Yaskawa INFORM job: X2_242(90,180).JBI

/JOB
//NAME X2_242(90,180)
///FOLDERNAME X2
//POS
///NPOS 135,135,135,3,0,0
///TOOL 0
///POSTYPE PULSE
///PULSE
C00000=-2000,-130321,-133031,0,28968,0
C00001=-117091,-130321,-133031,2123,28968,-3391
C00002=-159919,-130321,-133031,2123,28968,-3391
C00003=-159919,-130321,-133031,2123,87939,-3391
C00004=-105022,-108859,-78959,-31083,72176,-68730
C00005=-151007,-25092,-39063,-12800,65605,78235
C00006=-132593,67036,12002,-14068,96381,18620
C00007=-133669,66493,21901,-13656,90017,18991
C00008=-134090,67791,24612,-13544,88977,18967
C00009=-134090,67273,25686,-13543,88075,19066
C00010=-134090,67791,24612,-13544,88977,18967
C00011=-134073,67330,25416,-13547,88268,19050
C00012=-134739,69521,27996,-13380,87713,18892
C00013=-134073,67330,25416,-13547,88268,19050
C00014=-132576,62954,16151,-13952,91863,19138
C00015=-158058,56370,5063,-6789,93126,-12165
C00016=-161492,61731,13256,-13118,78465,-26852
C00017=-161219,65846,21027,-13360,75906,-26484
C00018=-161113,67624,24299,-13466,74851,-26332
C00019=-161114,67102,25367,-13521,73950,-26231
C00020=-161163,66904,24770,-13484,74201,-26276
C00021=-160433,68822,27026,-13824,73925,-25997
C00022=-161163,66904,24770,-13484,74201,-26276
C00023=-161111,67182,25269,-13516,74049,-26241
C00024=-161656,69750,28292,-13313,73437,-26358
C00025=-161111,67182,25269,-13516,74049,-26241
C00026=-161490,61134,14077,-13154,77673,-26766
C00027=-156757,36958,-7461,-10431,80488,-32893
C00028=-156267,40068,-956,-10702,78181,-32538
C00029=-156253,41350,1581,-10739,77295,-32458
C00030=-163911,62406,19268,6086,89764,-33901
C00031=-164446,59700,16177,9989,92313,-36673
C00032=-164418,59610,16075,9984,92326,-36663
C00033=-161961,50915,7130,7396,91423,-24195
C00034=-156779,43944,226,1104,89071,-15308
C00035=-150790,45819,2072,-7115,89912,-6230
C00036=-145239,57854,15312,-8608,88471,-4374
C00037=-145092,58025,15712,-8678,88333,-4325
C00038=-139841,72267,32142,-17294,91315,7524
C00039=-140946,99356,62874,-12757,94092,30974
C00040=-141208,101673,65869,-12719,93415,30955
C00041=-122713,94046,59869,-28177,93377,67521
C00042=-121487,97083,60557,-28349,94790,67637
C00043=-133468,48615,1742,-18804,93124,11842
C00044=-157997,71741,26694,-3661,70569,-66185
C00045=-156653,80960,41725,-4466,66130,-65572
C00046=-160707,58811,27097,7838,50776,-65613
C00047=-161862,58527,28132,10661,48808,-66136
C00048=-162060,71887,38599,9565,55625,-66013
C00049=-162634,67727,36532,11016,51381,-65293
C00050=-160821,61019,33044,3636,43624,-62105
C00051=-154148,75334,40185,-14517,57905,-63097
C00052=-154196,71820,32295,-14055,60854,-63507
C00053=-153288,55034,31796,-23088,50010,-69293
C00054=-151031,57353,45940,-40148,40347,-64995
C00055=-150621,58129,46816,-40537,40429,-64769
C00056=-149751,55668,48450,-47014,34319,-61006
C00057=-150747,54467,47461,-43008,31230,-60446
C00058=-154056,49858,42858,-29251,25609,-68749
C00059=-154872,47959,37614,-21306,28921,-70888
C00060=-159207,48403,28271,-1768,40383,-74494
C00061=-149846,52946,33243,-13952,46682,-81563
C00062=-149940,61587,46564,-14806,43022,-81015
C00063=-146336,59430,51340,-33146,36492,-77110
C00064=-145282,69746,63346,-35645,35179,-75711
C00065=-143319,74757,70706,-41882,34093,-73425
C00066=-141946,81470,79320,-45365,33350,-71705
C00067=-140704,87470,87386,-49528,32633,-69847
C00068=-140891,72507,62697,-35215,38758,-74780
C00069=-145179,75875,59784,-18821,43244,-78638
C00070=-151007,-25092,-39063,-12800,65605,78235
C00071=-105022,-108859,-78959,-31083,72176,-68730
C00072=-159919,-130321,-133031,2123,87939,-3391
C00073=-159919,-130321,-133031,2123,28968,-3391
C00074=-117091,-130321,-133031,2123,28968,-3391
C00075=31465,-130321,-133031,2123,28968,-3391
C00076=31465,-130321,-133031,2123,28968,-3391
C00077=70388,-93367,-87979,22259,92531,-40632
C00078=132234,14944,-6259,12342,59781,-23208
C00079=146205,63473,16177,10072,90044,-15024
C00080=148576,68007,22640,9405,88157,-14412
C00081=148576,67267,23954,9407,86985,-14500
C00082=148576,66783,24956,9411,86132,-14562
C00083=148576,66832,24863,9408,86216,-14555
C00084=149047,69084,27509,9276,85699,-14442
C00085=148423,68574,25700,9447,86607,-14574
C00086=146195,62986,16971,10071,89317,-15086
C00087=176137,58081,9771,-3198,80109,33161
C00088=174052,65626,21441,-2357,76742,32574
C00089=173571,63404,20046,-2157,76447,32425
C00090=173571,63211,20421,-2158,76117,32429
C00091=173571,63292,20263,-2157,76255,32427
C00092=172556,64401,21545,-1729,76012,32099
C00093=173019,62971,18478,-1917,77173,32231
C00094=167045,54371,14180,12829,67421,32117
C00095=167300,57261,17419,12739,66888,32149
C00096=166775,56105,16119,12998,67167,31995
C00097=174959,61653,15361,-2721,78467,32830
C00098=153862,58220,7137,12336,84382,31788
C00099=154888,58914,9595,11964,83110,31986
C00100=146416,53637,12500,29969,73855,35683
C00101=161804,89703,42514,-6671,93266,37768
C00102=160481,83040,34267,-6425,94812,37264
C00103=160461,82996,34213,-6421,94821,37257
C00104=160314,82402,33477,-6393,94958,37204
C00105=155818,71683,20777,1425,95566,24197
C00106=154068,75736,24755,2435,97986,16967
C00107=150406,78568,28210,7412,98870,8330
C00108=143192,78361,31098,15429,92978,3071
C00109=142524,84239,37703,11837,92418,-12035
C00110=142502,84415,37922,11841,92377,-12046
C00111=137937,102743,61702,17663,90401,-30375
C00112=138214,107970,68255,17604,89055,-30475
C00113=138254,108650,69203,17597,88823,-30493
C00114=137728,105908,62856,17713,91318,-30315
C00115=129809,68648,23314,23742,79294,-62187
C00116=130521,38108,-11366,22924,75116,-53839
C00117=144715,56131,10361,11744,72134,27543
C00118=151566,59831,28742,-2859,46138,64220
C00119=152051,66365,37606,-3402,44065,64516
C00120=152470,67516,39026,-3796,43800,64724
C00121=153239,74187,48057,-1867,40213,65616
C00122=151811,68486,39030,4846,43626,66812
C00123=148976,61300,30711,7226,45253,65595
C00124=147729,58500,33654,14300,37151,64277
C00125=144430,59667,36614,25817,36412,63257
C00126=144460,72482,45840,17180,42284,64323
C00127=143111,63918,40413,22730,36091,62179
C00128=143801,66633,41900,20305,38275,63153
C00129=139817,77107,57238,29606,33210,58883
C00130=141383,82478,55565,14874,41935,61497
C00131=144692,57703,21103,13544,52726,73165
C00132=140496,9250,-2578,20724,48099,77689
C00133=103999,-84119,-66645,26288,35960,55555
C00134=-2000,-130321,-133031,0,28968,0
BC00000=147972,491577,1075193
BC00001=188398,1906,1075193
BC00002=367644,-164195,1075193
BC00003=367644,-172087,1075193
BC00004=367644,-179096,239389
BC00005=367644,-179096,202799
BC00006=311795,-165148,45027
BC00007=311795,-165148,45027
BC00008=311795,-165148,45027
BC00009=311795,-165148,45027
BC00010=311795,-165148,45027
BC00011=311795,-165148,45027
BC00012=311795,-165148,45027
BC00013=311795,-165148,45027
BC00014=311795,-165148,45027
BC00015=362414,-140809,31779
BC00016=380271,-154677,8218
BC00017=380271,-154677,8218
BC00018=380271,-154677,8218
BC00019=380271,-154677,8218
BC00020=380271,-154677,8218
BC00021=380271,-154677,8218
BC00022=380271,-154677,8218
BC00023=380271,-154677,8218
BC00024=380271,-154677,8218
BC00025=380271,-154677,8218
BC00026=380271,-154677,8218
BC00027=343072,-138712,53288
BC00028=343072,-138712,53288
BC00029=343072,-138712,53288
BC00030=343072,-138712,53288
BC00031=343072,-138713,53287
BC00032=343072,-138713,53287
BC00033=343072,-138712,53288
BC00034=343072,-138712,53286
BC00035=343072,-138712,53286
BC00036=343072,-138712,53286
BC00037=343072,-138712,53284
BC00038=343072,-138712,53286
BC00039=343072,-138712,53286
BC00040=343072,-138712,53286
BC00041=294648,-138712,53288
BC00042=294648,-138712,53288
BC00043=320422,-160767,40892
BC00044=369045,-176137,27013
BC00045=367905,-178617,27013
BC00046=367905,-178910,27013
BC00047=367905,-178910,27013
BC00048=367905,-179959,27013
BC00049=367905,-180015,27013
BC00050=367905,-179162,27013
BC00051=367905,-179037,27013
BC00052=367905,-178812,27013
BC00053=384322,-166528,125648
BC00054=384322,-166528,125648
BC00055=384322,-166528,125648
BC00056=384322,-166528,125648
BC00057=384322,-166528,125648
BC00058=384322,-166528,125648
BC00059=384322,-166528,125648
BC00060=384322,-166528,125648
BC00061=367644,-168516,156611
BC00062=367644,-172191,156611
BC00063=367644,-171321,156611
BC00064=367644,-179096,156611
BC00065=367644,-179096,156611
BC00066=367644,-179096,156611
BC00067=367644,-179096,156611
BC00068=367644,-179096,156611
BC00069=367644,-179096,156611
BC00070=367644,-179096,202799
BC00071=367644,-179096,239389
BC00072=367644,-179096,1075193
BC00073=367644,-179096,1075193
BC00074=188398,1906,1075193
BC00075=341060,491577,1075193
BC00076=341060,491577,1075193
BC00077=258990,522046,241931
BC00078=356760,522046,241931
BC00079=356760,409759,42887
BC00080=356760,409759,42887
BC00081=356760,409759,42887
BC00082=356760,409759,42887
BC00083=356760,409759,42887
BC00084=356760,409759,42887
BC00085=356760,409759,42887
BC00086=356760,409759,42887
BC00087=398158,391605,17411
BC00088=398158,391605,17411
BC00089=398158,391605,17411
BC00090=398158,391605,17411
BC00091=398158,391605,17411
BC00092=398158,391605,17411
BC00093=398158,391605,17411
BC00094=398158,391605,17411
BC00095=398158,391605,17411
BC00096=398158,391605,17411
BC00097=398158,391605,17411
BC00098=344176,409815,17
BC00099=344176,409815,17
BC00100=344176,409815,17
BC00101=344176,409815,17
BC00102=344176,409815,17
BC00103=344176,409815,17
BC00104=344176,409815,17
BC00105=344176,409815,15
BC00106=344176,409815,17
BC00107=344176,409815,17
BC00108=344176,409815,13
BC00109=344176,409815,12
BC00110=344176,409815,12
BC00111=344176,409815,12
BC00112=344176,409815,12
BC00113=344176,409815,12
BC00114=344176,409815,12
BC00115=326504,409815,17
BC00116=326504,409815,17
BC00117=339270,441939,17014
BC00118=344994,456339,24633
BC00119=344994,456339,24633
BC00120=344994,456339,24633
BC00121=344994,456339,24633
BC00122=344994,456339,24631
BC00123=344994,456339,24631
BC00124=344994,456339,24631
BC00125=344994,456339,24631
BC00126=344994,456339,24631
BC00127=344994,456339,24631
BC00128=344994,456339,24631
BC00129=344994,456339,24631
BC00130=344994,456339,24631
BC00131=359830,449275,49809
BC00132=372188,522287,309305
BC00133=335727,515780,471592
BC00134=200118,491577,1075193
EC00000=-798156,-1296783
EC00001=-798156,-1296783
EC00002=-798156,-1296783
EC00003=-798156,-1296783
EC00004=-798156,-1296783
EC00005=-798156,-1296783
EC00006=-798156,-1296783
EC00007=-798156,-1296783
EC00008=-798156,-1296783
EC00009=-798156,-1296783
EC00010=-798156,-1296783
EC00011=-798156,-1296783
EC00012=-798156,-1296783
EC00013=-798156,-1296783
EC00014=-798156,-1296783
EC00015=-798156,-1296783
EC00016=-798156,-1296783
EC00017=-798156,-1296783
EC00018=-798156,-1296783
EC00019=-798156,-1296783
EC00020=-798156,-1296783
EC00021=-798156,-1296783
EC00022=-798156,-1296783
EC00023=-798156,-1296783
EC00024=-798156,-1296783
EC00025=-798156,-1296783
EC00026=-798156,-1296783
EC00027=-798156,-1296783
EC00028=-798156,-1296783
EC00029=-798156,-1296783
EC00030=-798156,-1296783
EC00031=-798155,-1296782
EC00032=-798155,-1296782
EC00033=-798156,-1296783
EC00034=-798155,-1296782
EC00035=-798155,-1296782
EC00036=-798155,-1296782
EC00037=-798155,-1296781
EC00038=-798155,-1296782
EC00039=-798155,-1296782
EC00040=-798155,-1296782
EC00041=-798156,-1296783
EC00042=-798156,-1296783
EC00043=-798156,-1296783
EC00044=-798156,-1296783
EC00045=-798156,-1296783
EC00046=-798156,-1296783
EC00047=-798156,-1296783
EC00048=-798156,-1296783
EC00049=-798156,-1296783
EC00050=-798156,-1296783
EC00051=-798156,-1296783
EC00052=-798156,-1296783
EC00053=-798156,-1296783
EC00054=-798156,-1296783
EC00055=-798156,-1296783
EC00056=-798156,-1296783
EC00057=-798156,-1296783
EC00058=-798156,-1296783
EC00059=-798156,-1296783
EC00060=-798156,-1296783
EC00061=-798156,-1296783
EC00062=-798156,-1296783
EC00063=-798156,-1296783
EC00064=-798156,-1296783
EC00065=-798156,-1296783
EC00066=-798156,-1296783
EC00067=-798156,-1296783
EC00068=-798156,-1296783
EC00069=-798156,-1296783
EC00070=-798156,-1296783
EC00071=-798156,-1296783
EC00072=-798156,-1296783
EC00073=-798156,-1296783
EC00074=-798156,-1296783
EC00075=-798156,-1296783
EC00076=798156,-1296783
EC00077=798156,-1296783
EC00078=798156,-1296783
EC00079=798156,-1296783
EC00080=798156,-1296783
EC00081=798156,-1296783
EC00082=798156,-1296783
EC00083=798156,-1296783
EC00084=798156,-1296783
EC00085=798156,-1296783
EC00086=798156,-1296783
EC00087=798156,-1296783
EC00088=798156,-1296783
EC00089=798156,-1296783
EC00090=798156,-1296783
EC00091=798156,-1296783
EC00092=798156,-1296783
EC00093=798156,-1296783
EC00094=798156,-1296783
EC00095=798156,-1296783
EC00096=798156,-1296783
EC00097=798156,-1296783
EC00098=798156,-1296783
EC00099=798156,-1296783
EC00100=798156,-1296783
EC00101=798156,-1296783
EC00102=798156,-1296783
EC00103=798156,-1296783
EC00104=798156,-1296783
EC00105=798155,-1296783
EC00106=798156,-1296783
EC00107=798156,-1296783
EC00108=798154,-1296784
EC00109=798154,-1296784
EC00110=798154,-1296784
EC00111=798154,-1296784
EC00112=798154,-1296784
EC00113=798154,-1296784
EC00114=798154,-1296784
EC00115=798156,-1296783
EC00116=798156,-1296783
EC00117=798156,-1296783
EC00118=798155,-1296783
EC00119=798155,-1296783
EC00120=798155,-1296783
EC00121=798155,-1296783
EC00122=798154,-1296784
EC00123=798154,-1296784
EC00124=798154,-1296784
EC00125=798154,-1296784
EC00126=798154,-1296784
EC00127=798154,-1296784
EC00128=798154,-1296784
EC00129=798154,-1296784
EC00130=798154,-1296784
EC00131=798155,-1296783
EC00132=798155,-1296783
EC00133=798155,-1296783
EC00134=798156,-1296783
///POSTYPE BASE
///RECTAN
///RCONF 0,0,0,0,1,0,0,0,0,0,0,0,0,0,0,0,0,0,0,0,0,0,0,0
P00006=2.006,1.622,-0.565,0.0000,0.0000,0.0000
P00021=0.073,2.058,-0.109,0.0000,0.0000,0.0000
P00022=2.006,1.622,-0.565,0.0000,0.0000,0.0000
//INST
///DATE 2024/11/26 22:05
///ATTR SC,RW
///GROUP1 RB1,BS1
///GROUP2 ST1
NOP
'X2_242(90,180)
'-90,0
MOVJ C00000 BC00000 VJ=100.00  +MOVJ EC00000 VJ=100.00
MOVJ C00001 BC00001 VJ=80.00  +MOVJ EC00001 VJ=100.00
MOVJ C00002 BC00002 VJ=70.00  +MOVJ EC00002 VJ=100.00
MOVJ C00003 BC00003 VJ=100.00  +MOVJ EC00003 VJ=100.00
MOVJ C00004 BC00004 VJ=100.00  +MOVJ EC00004 VJ=100.00
MOVJ C00005 BC00005 VJ=100.00  +MOVJ EC00005 VJ=100.00
'Path S4220
SFTOF3D
MOVJ C00006 BC00006 VJ=100.00  +MOVJ EC00006 VJ=100.00
MOVL C00007 BC00007 V=666.7  +MOVJ EC00007 VJ=100.00
SMOVL C00008 BC00008 V=166.7  +MOVJ EC00008
SREFP 3 C00009 BC00009  +REFP EC00009
CALL JOB:SEARCH-R1-S13D
SET P022 P006
SFTON3D P022
SMOVL C00010 BC00010 V=166.7  +MOVJ EC00010
SMOVL C00011 BC00011 V=166.7  +MOVJ EC00011
SREFP 3 C00012 BC00012  +REFP EC00012
CALL JOB:SEARCH-R1-S13D
SET P022 P006
SFTON3D P022
SMOVL C00013 BC00013 V=166.7  +MOVJ EC00013
MOVL C00014 BC00014 V=1000.0  +MOVJ EC00014 VJ=100.00
'EndPath S4220
MOVJ C00015 BC00015 VJ=100.00  +MOVJ EC00015 VJ=100.00
'Path S3549
SFTOF3D
MOVJ C00016 BC00016 VJ=100.00  +MOVJ EC00016 VJ=100.00
MOVL C00017 BC00017 V=666.7  +MOVJ EC00017 VJ=100.00
SMOVL C00018 BC00018 V=166.7  +MOVJ EC00018
SREFP 3 C00019 BC00019  +REFP EC00019
CALL JOB:SEARCH-R1-S13D
SET P021 P006
SFTON3D P021
SMOVL C00020 BC00020 V=166.7  +MOVJ EC00020
SREFP 3 C00021 BC00021  +REFP EC00021
CALL JOB:SEARCH-R1-S13D
SET P021 P006
SFTON3D P021
SMOVL C00022 BC00022 V=166.7  +MOVJ EC00022
SMOVL C00023 BC00023 V=166.7  +MOVJ EC00023
SREFP 3 C00024 BC00024  +REFP EC00024
CALL JOB:SEARCH-R1-S13D
SET P021 P006
SFTON3D P021
SMOVL C00025 BC00025 V=166.7  +MOVJ EC00025
MOVL C00026 BC00026 V=1000.0  +MOVJ EC00026 VJ=100.00
'EndPath S3549
'Path W3550
SFTOF3D
SSFTOF
SFTOF
SFTON3D P021
MOVJ C00027 BC00027 VJ=100.00  +MOVJ EC00027 VJ=100.00
SMOVL C00028 BC00028 V=666.7  +MOVJ EC00028
SMOVL C00029 BC00029 V=166.7 PL=0  +MOVJ EC00029
MACRO1 MJ#(0) ARGF9
ARCON
SMOVL C00030 BC00030 V=8.3  +MOVJ EC00030
SMOVL C00031 BC00031 V=8.3  +MOVJ EC00031
SMOVC C00032 BC00032 V=10.0  +MOVJ EC00032
SMOVC C00033 BC00033 V=10.0  +MOVJ EC00033
SFTON3D P022
SMOVC C00034 BC00034 V=10.0  +MOVJ EC00034
SMOVC C00035 BC00035 V=10.0  +MOVJ EC00035
SMOVL C00036 BC00036 V=10.0  +MOVJ EC00036
SFTON3D P021
SMOVC C00037 BC00037 V=10.0  +MOVJ EC00037
SMOVC C00038 BC00038 V=10.0  +MOVJ EC00038
SMOVC C00039 BC00039 V=10.0  +MOVJ EC00039
SMOVC C00040 BC00040 V=8.3  +MOVJ EC00040
ARCOF
SMOVL C00041 BC00041 V=800.0  +MOVJ EC00041
SMOVL C00042 BC00042 V=1000.0  +MOVJ EC00042
SFTOF3D
'EndPath W3550
MOVJ C00043 BC00043 VJ=100.00  +MOVJ EC00043 VJ=100.00
'Path W3552
SFTOF3D
SFTON3D P021
MOVJ C00044 BC00044 VJ=100.00  +MOVJ EC00044 VJ=100.00
SMOVL C00045 BC00045 V=800.0  +MOVJ EC00045
SMOVL C00046 BC00046 V=166.7  +MOVJ EC00046
MACRO1 MJ#(0) ARGF21
ARCON
SMOVL C00047 BC00047 V=9.2  +MOVJ EC00047
SMOVL C00048 BC00048 V=9.2  +MOVJ EC00048
SMOVL C00049 BC00049 V=9.2  +MOVJ EC00049
SMOVL C00050 BC00050 V=9.2  +MOVJ EC00050
ARCOF
SMOVL C00051 BC00051 V=800.0  +MOVJ EC00051
SMOVL C00052 BC00052 V=1000.0  +MOVJ EC00052
SFTOF3D
'EndPath W3552
'Path W3553
SFTOF3D
SFTON3D P022
MOVJ C00053 BC00053 VJ=100.00  +MOVJ EC00053 VJ=100.00
SMOVL C00054 BC00054 V=166.7 PL=0  +MOVJ EC00054
ARCON
SMOVL C00055 BC00055 V=8.3  +MOVJ EC00055
SMOVL C00056 BC00056 V=8.3  +MOVJ EC00056
SMOVL C00057 BC00057 V=8.3  +MOVJ EC00057
SMOVL C00058 BC00058 V=8.3  +MOVJ EC00058
ARCOF
SMOVL C00059 BC00059 V=800.0  +MOVJ EC00059
SMOVL C00060 BC00060 V=1000.0  +MOVJ EC00060
SFTOF3D
'EndPath W3553
'Path W3554
SFTOF3D
SFTON3D P022
MOVJ C00061 BC00061 VJ=50.00  +MOVJ EC00061 VJ=100.00
SMOVL C00062 BC00062 V=500.0  +MOVJ EC00062
SMOVL C00063 BC00063 V=166.7 PL=0  +MOVJ EC00063
ARCON
SMOVL C00064 BC00064 V=8.3  +MOVJ EC00064
SMOVL C00065 BC00065 V=8.3  +MOVJ EC00065
SMOVL C00066 BC00066 V=8.3  +MOVJ EC00066
SMOVL C00067 BC00067 V=8.3  +MOVJ EC00067
ARCOF
SMOVL C00068 BC00068 V=800.0  +MOVJ EC00068
SMOVL C00069 BC00069 V=1000.0  +MOVJ EC00069
SFTOF3D
'EndPath W3554
MOVJ C00070 BC00070 VJ=100.00  +MOVJ EC00070 VJ=100.00
MOVJ C00071 BC00071 VJ=100.00  +MOVJ EC00071 VJ=100.00
MOVJ C00072 BC00072 VJ=100.00  +MOVJ EC00072 VJ=100.00
MOVJ C00073 BC00073 VJ=100.00  +MOVJ EC00073 VJ=100.00
MOVJ C00074 BC00074 VJ=100.00  +MOVJ EC00074 VJ=100.00
MOVJ C00075 BC00075 VJ=100.00  +MOVJ EC00075 VJ=100.00
MOVJ C00076 BC00076 VJ=100.00  +MOVJ EC00076 VJ=100.00
'-90,180
CALL JOB:CLEAN-R1_KM_NEW
MOVJ C00077 BC00077 VJ=100.00  +MOVJ EC00077 VJ=100.00
MOVJ C00078 BC00078 VJ=100.00  +MOVJ EC00078 VJ=100.00
'Path S4222
SFTOF3D
MOVJ C00079 BC00079 VJ=100.00  +MOVJ EC00079 VJ=100.00
MOVL C00080 BC00080 V=666.7  +MOVJ EC00080 VJ=100.00
SMOVL C00081 BC00081 V=166.7  +MOVJ EC00081
SREFP 3 C00082 BC00082  +REFP EC00082
CALL JOB:SEARCH-R1-S13D
SET P022 P006
SFTON3D P022
SMOVL C00083 BC00083 V=166.7  +MOVJ EC00083
SREFP 3 C00084 BC00084  +REFP EC00084
CALL JOB:SEARCH-R1-S13D
SET P022 P006
SFTON3D P022
SMOVL C00085 BC00085 V=166.7  +MOVJ EC00085
SFTOF3D
MOVL C00086 BC00086 V=1000.0  +MOVJ EC00086 VJ=100.00
'EndPath S4222
'Path S4223
SFTOF3D
MOVJ C00087 BC00087 VJ=100.00  +MOVJ EC00087 VJ=100.00
MOVL C00088 BC00088 V=666.7  +MOVJ EC00088 VJ=100.00
SMOVL C00089 BC00089 V=166.7  +MOVJ EC00089
SREFP 3 C00090 BC00090  +REFP EC00090
CALL JOB:SEARCH-R1-S13D
SET P021 P006
SFTON3D P021
SMOVL C00091 BC00091 V=166.7  +MOVJ EC00091
SREFP 3 C00092 BC00092  +REFP EC00092
CALL JOB:SEARCH-R1-S13D
SET P021 P006
SFTON3D P021
SMOVL C00093 BC00093 V=166.7  +MOVJ EC00093
SMOVL C00094 BC00094 V=166.7  +MOVJ EC00094
SREFP 3 C00095 BC00095  +REFP EC00095
CALL JOB:SEARCH-R1-S13D
SET P021 P006
SFTON3D P021
SMOVL C00096 BC00096 V=166.7  +MOVJ EC00096
MOVL C00097 BC00097 V=1000.0  +MOVJ EC00097 VJ=100.00
'EndPath S4223
'Path W4224
SFTOF3D
MOVJ C00098 BC00098 VJ=100.00  +MOVJ EC00098 VJ=100.00
SFTON3D P021
MOVL C00099 BC00099 V=666.7  +MOVJ EC00099 VJ=100.00
SMOVL C00100 BC00100 V=166.7 PL=0  +MOVJ EC00100
MACRO1 MJ#(0) ARGF9
ARCON
SMOVL C00101 BC00101 V=10.0  +MOVJ EC00101
SMOVL C00102 BC00102 V=9.2  +MOVJ EC00102
SMOVC C00103 BC00103 V=10.0  +MOVJ EC00103
SMOVC C00104 BC00104 V=10.0  +MOVJ EC00104
SFTON3D P022
SMOVC C00105 BC00105 V=10.0  +MOVJ EC00105
SMOVC C00106 BC00106 V=10.0  +MOVJ EC00106
SMOVC C00107 BC00107 V=10.0  +MOVJ EC00107
SMOVL C00108 BC00108 V=10.0  +MOVJ EC00108
SMOVL C00109 BC00109 V=10.0  +MOVJ EC00109
SMOVC C00110 BC00110 V=9.2  +MOVJ EC00110
SFTON3D P021
SMOVC C00111 BC00111 V=10.0  +MOVJ EC00111
SMOVC C00112 BC00112 V=10.0  +MOVJ EC00112
SMOVL C00113 BC00113 V=10.0  +MOVJ EC00113
ARCOF
MOVL C00114 BC00114 V=800.0  +MOVJ EC00114 VJ=100.00
MOVL C00115 BC00115 V=1000.0  +MOVJ EC00115 VJ=100.00
'EndPath W4224
MOVJ C00116 BC00116 VJ=100.00  +MOVJ EC00116 VJ=100.00
MOVJ C00117 BC00117 VJ=100.00  +MOVJ EC00117 VJ=100.00
'Path W4225
SFTOF3D
SFTON3D P021
SMOVL C00118 BC00118 V=800.0  +MOVJ EC00118
SMOVL C00119 BC00119 V=166.7 PL=0  +MOVJ EC00119
MACRO1 MJ#(0) ARGF21
ARCON
SMOVL C00120 BC00120 V=7.5  +MOVJ EC00120
SMOVL C00121 BC00121 V=7.5  +MOVJ EC00121
ARCOF
SMOVL C00122 BC00122 V=800.0  +MOVJ EC00122
SMOVL C00123 BC00123 V=1000.0  +MOVJ EC00123
SFTOF3D
'EndPath W4225
'Path W4226
SFTOF3D
SFTON3D P022
SMOVL C00124 BC00124 V=166.7 PL=0  +MOVJ EC00124
ARCON
SMOVL C00125 BC00125 V=8.3  +MOVJ EC00125
SMOVL C00126 BC00126 V=8.3  +MOVJ EC00126
ARCOF
SMOVL C00127 BC00127 V=800.0  +MOVJ EC00127
SFTOF3D
'EndPath W4226
'Path W4227
SFTOF3D
SFTON3D P022
SMOVL C00128 BC00128 V=166.7 PL=0  +MOVJ EC00128
ARCON
SMOVL C00129 BC00129 V=7.5  +MOVJ EC00129
ARCOF
SMOVL C00130 BC00130 V=800.0  +MOVJ EC00130
SMOVL C00131 BC00131 V=1000.0  +MOVJ EC00131
SFTOF3D
'EndPath W4227
MOVJ C00132 BC00132 VJ=100.00  +MOVJ EC00132 VJ=100.00
MOVJ C00133 BC00133 VJ=100.00  +MOVJ EC00133 VJ=100.00
MOVJ C00134 BC00134 VJ=100.00  +MOVJ EC00134 VJ=100.00
END
